ABB RobotStudio station: Tehtävä 18 Smart_Component_20230512-152205.rsstn

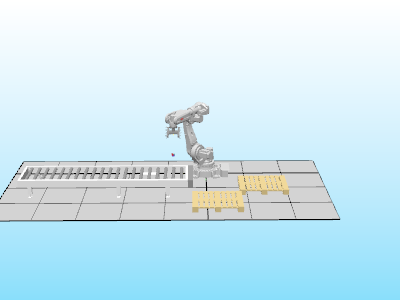
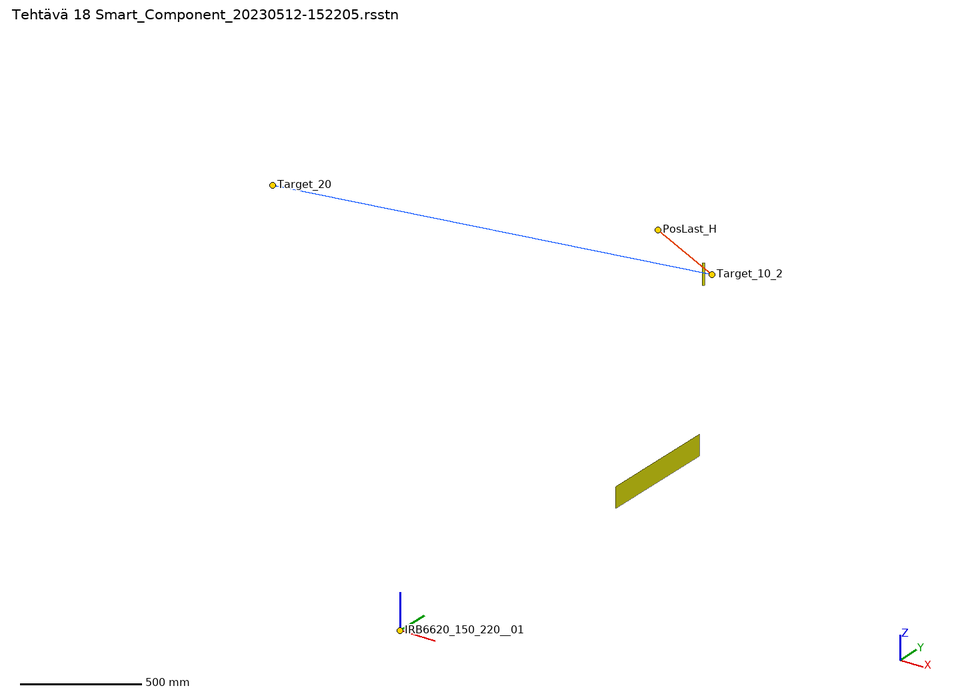
[picture v1: parts stored in the station drawn from their meshes, with robot base, taught points and paths (robot models come from the ABB library and are not in the file)]
Station SmartComponentProject_5_TEST (saved by RobotStudio 22.3.10141.1)
Controller SmartComponentTest
  mechanical unit ROB_1: IRB6620_150_220__01, 6 joints, base frame (0, 0, 0) mm
Layout (positions relative to the parent item):
  - IRB6620_150_220__01 [mechanism, from Robots\IRB6620_150_220_G_01.rslib] at (0, 0, 0) mm; joint values [1.1039, 0.1854, -0.0725, 0, 1.4578, -2.0377] (rad or m)
  - euro_pallet [part, from Libraries\euro_pallet.rslib] at (-855.44, 1560.26, 0) mm
  - euro [part, from Libraries\euro_pallet.rslib] at (-2029.52, 494.94, 0) mm
  - Syöttökuljetin [smart component]
      signals: DO BOX_POS, DI STOP
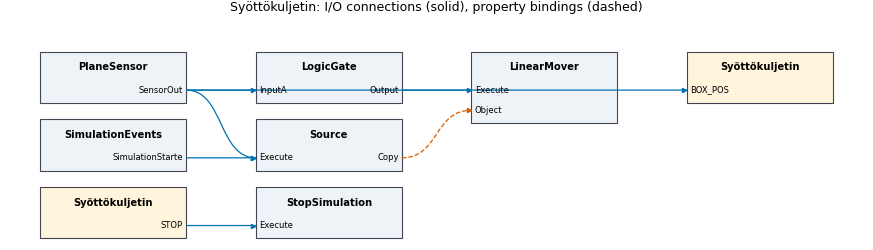
      connections:
        PlaneSensor.SensorOut -> Syöttökuljetin.BOX_POS
        LogicGate.Output -> LinearMover.Execute
        PlaneSensor.SensorOut -> LogicGate.InputA
        PlaneSensor.SensorOut -> Source.Execute
        SimulationEvents.SimulationStarted -> Source.Execute
        Syöttökuljetin.STOP -> StopSimulation.Execute
        Source.Copy => LinearMover.Object
    - Kuljetin [part, from Equipment\Conveyor 950 4000 h2.rslib] at (450, 600, 0) mm
    - LinearMover [smart component, from Components\LinearMover.rslib]
        properties: Object=(none); Direction=[-1 0 0]; Speed=0.5; Reference=Global; ReferenceObject=(none)
    - Source [smart component, from Components\Source.rslib] at (-9000, 0, 0) mm
        properties: Source=Laatikko; Copy=(none); Parent=(none); Position=[0 0 0]; Orientation=[0 0 0]; Transient=false; PhysicsBehavior=0
    - PlaneSensor [smart component, from Components\PlaneSensor.rslib] at (555.57, 745.74, 515.06) mm, rotated rx 0 ry 90 rz 0 deg
        properties: Origin=[0 0 0]; Axis1=[0.1 0 0]; Axis2=[0 0.6 0]; SensedPart=(none)
      - _sensorPart_ [part], size 100 x 600 x 0 mm
    - Laatikko [part], size 500 x 500 x 500 mm
    - LogicGate [smart component, from Components\LogicGate.rslib]
        properties: Operator=NOT; Delay=0
    - SimulationEvents [smart component, from Components\SimulationEvents.rslib]
    - StopSimulation [smart component, from Components\StopSimulation.rslib]
  - Tarttuja [smart component]
      signals: DI pudota, DI pida_laatikkoa, DO Laatikko_Kourassa, DI destroy
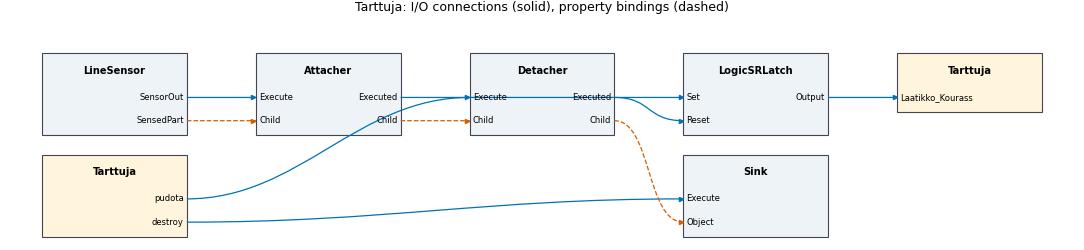
      connections:
        LineSensor.SensorOut -> Attacher.Execute
        Tarttuja.pudota -> Detacher.Execute
        Attacher.Executed -> LogicSRLatch.Set
        Detacher.Executed -> LogicSRLatch.Reset
        LogicSRLatch.Output -> Tarttuja.Laatikko_Kourassa
        Tarttuja.destroy -> Sink.Execute
        LineSensor.SensedPart => Attacher.Child
        Attacher.Child => Detacher.Child
        Detacher.Child => Sink.Object
    - VacuumGripper [mechanism, from Libraries\VacuumGripper.rslib] at (801.58, 1086.46, 1611.5) mm, rotated rx 180 ry 0 rz 0 deg
    - Attacher [smart component, from Components\Attacher.rslib]
        properties: Parent=VacuumGripper; Flange=0; Child=(none); Mount=false; Offset=[0 0 0]; Orientation=[0 0 0]
    - Detacher [smart component, from Components\Detacher.rslib]
        properties: Child=(none); KeepPosition=true
    - LineSensor [smart component, from Components\LineSensor.rslib] at (801.58, 1023.02, 1492.8) mm, rotated rx 180 ry 0 rz 0 deg
        properties: Start=[0 0 0]; End=[0 0 0.1]; Radius=0.005; SensedPart=(none); SensedPoint=[0 0 0]
      - _sensorPart_ [part], size 10 x 10 x 100 mm
    - LogicSRLatch [smart component, from Components\LogicSRLatch.rslib]
    - Sink [smart component, from Components\Sink.rslib]
        properties: Object=(none)
  - Frame_1 [frame] at (801.58, 1086.46, 914) mm, rotated rx 180 ry 0 rz 0 deg
Attachment: VacuumGripper is attached to IRB6620_150_220__01 / Link6
Attachment: LineSensor is attached to VacuumGripper / vacuum_gripper
Attachment: Source is attached to Laatikko
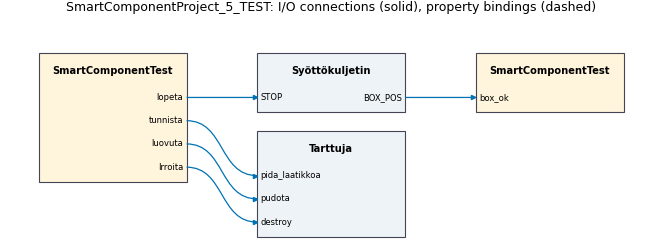
Station logic (signal -> signal, property => property):
  SmartComponentTest.lopeta -> Syöttökuljetin.STOP
  Syöttökuljetin.BOX_POS -> SmartComponentTest.box_ok
  SmartComponentTest.tunnista -> Tarttuja.pida_laatikkoa
  SmartComponentTest.luovuta -> Tarttuja.pudota
  SmartComponentTest.Irroita -> Tarttuja.destroy
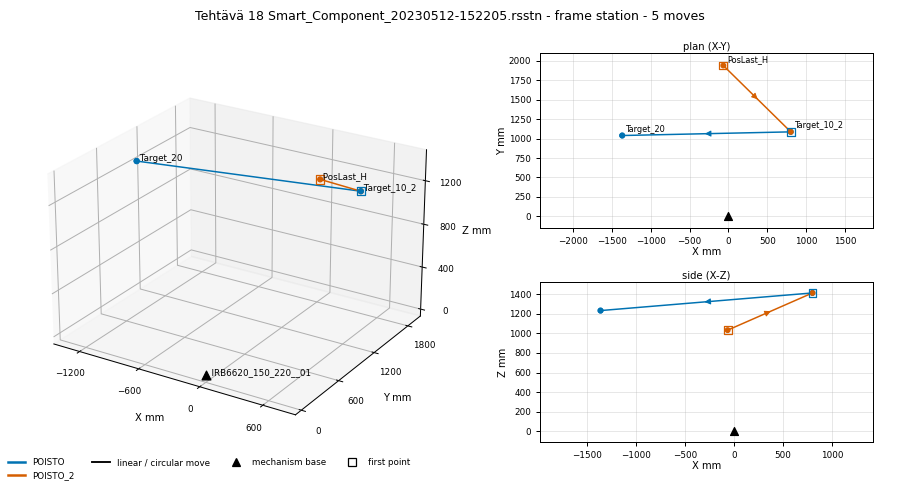
[picture p0: tool path of Tehtävä 18 Smart_Component_20230512-152205.rsstn in frame station, 5 of 5 moves have a stored position in this frame; points joined in program order, loops and branches not executed]
Targets, tools, work objects and paths stored in the station, written as RAPID:
! task T_ROB1
MODULE CalibData
  PERS tooldata tGripper:=[TRUE,[[0,0,197.5],[1,0,0,0]],[25,[0,0.00109327,116.889],[1,0,0,0],0,0,0]];
  TASK PERS wobjdata Lava2:=[FALSE,TRUE,"",[[0,0,0],[1,0,0,0]],[[0,0,0],[1,0,0,0]]];
ENDMODULE

! task T_ROB1
MODULE Module1
  CONST robtarget Target_10_2:=[[801.58,1086.458,1414],[0,1,0,0],[0,0,-2,0],[9E+09,9E+09,9E+09,9E+09,9E+09,9E+09]];
  CONST robtarget Target_20:=[[-1365.910561248,1039.448894024,1233.637],[0,1,0,0],[1,0,-1,0],[9E+09,9E+09,9E+09,9E+09,9E+09,9E+09]];
  CONST robtarget PosLast_H:=[[-65.910561248,1939.448894024,1033.637],[0,1,0,0],[1,0,-1,0],[9E+09,9E+09,9E+09,9E+09,9E+09,9E+09]];
  CONST robtarget Pos_1_H:=[[801.58,1086.458,1414],[0,1,0,0],[0,0,-2,0],[9E+09,9E+09,9E+09,9E+09,9E+09,9E+09]];
  PROC POISTO()
    MoveL Target_10_2,v1000,z0,tool0\WObj:=wobj0;
    MoveL Target_20,v1000,z0,tGripper\WObj:=wobj0;
    WaitTime 0.1;
    WaitTime 0.1;
    MoveL Target_20,v1000,fine,tGripper\WObj:=wobj0;
  ENDPROC
  PROC main()
    SetDO lopeta,1;
    POISTO;
    POISTO_2;
  ENDPROC
  PROC POISTO_2()
    MoveL PosLast_H,v1000,z100,tGripper\WObj:=Lava2;
    WaitTime 0.1;
    WaitTime 0.1;
    MoveL Pos_1_H,v1000,z100,tGripper\WObj:=Lava2;
  ENDPROC
ENDMODULE

